# EPICS autosave request: calc/calcApp/Db/userCalcOuts10more_settings.req
file calcout_settings.req P=$(P)userCalcOut$(N1)
file calcout_settings.req P=$(P)userCalcOut$(N2)
file calcout_settings.req P=$(P)userCalcOut$(N3)
file calcout_settings.req P=$(P)userCalcOut$(N4)
file calcout_settings.req P=$(P)userCalcOut$(N5)
file calcout_settings.req P=$(P)userCalcOut$(N6)
file calcout_settings.req P=$(P)userCalcOut$(N7)
file calcout_settings.req P=$(P)userCalcOut$(N8)
file calcout_settings.req P=$(P)userCalcOut$(N9)
file calcout_settings.req P=$(P)userCalcOut$(N10)
